DATA_BLOCK "Elev"
{ S7_Optimized_Access := 'TRUE' }
VERSION : 0.1
NON_RETAIN
   VAR
      eet_autorun : Bool;   // 自动运行信号
      plc_ready : Bool;   // 准备就绪信号
      elev { S7_SetPoint := 'False'} : Array[1.."ELE_SUM"] of "Elevator_Class";   // 电梯序号
      btn_outside { S7_SetPoint := 'False'} : Array[1..2, 1.."FlOOR_TOP"] of "Button_Class";   // 公共外部按键
   END_VAR


BEGIN

END_DATA_BLOCK

